// TIA Portal V21 export
FUNCTION "Motore_CentrifugaLavaggio" : Void   // FC135, LAD
{ S7_Optimized_Access := 'TRUE' }
// stored: SetENOAutomatically false
   VAR_TEMP
      AutoPos : Bool;
      AutoNeg : Bool;
   END_VAR
BEGIN

REGION Network 1: Comando positivo in automatico
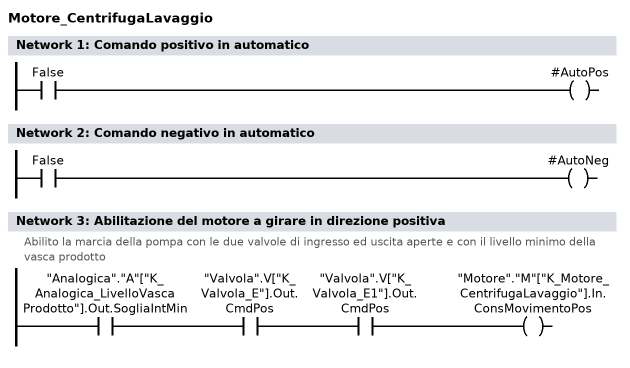
   RUNG wire#powerrail
      Contact( False )
      Coil( #AutoPos )
   END_RUNG
   // the same network as SCL:
   #AutoPos := False;
END_REGION

REGION Network 2: Comando negativo in automatico
   RUNG wire#powerrail
      Contact( False )
      Coil( #AutoNeg )
   END_RUNG
   // the same network as SCL:
   #AutoNeg := False;
END_REGION

REGION Network 3: Abilitazione del motore a girare in direzione positiva
   // Abilito la marcia della pompa con le due valvole di ingresso ed uscita aperte e con il livello minimo della vasca prodotto
   RUNG wire#powerrail
      Contact( "Analogica"."A"["K_Analogica_LivelloVascaProdotto"].Out.SogliaIntMin )
      Contact( "Valvola".V["K_Valvola_E"].Out.CmdPos )
      Contact( "Valvola".V["K_Valvola_E1"].Out.CmdPos )
      Coil( "Motore"."M"["K_Motore_CentrifugaLavaggio"].In.ConsMovimentoPos )
   END_RUNG
   // the same network as SCL:
   "Motore"."M"["K_Motore_CentrifugaLavaggio"].In.ConsMovimentoPos := "Analogica"."A"["K_Analogica_LivelloVascaProdotto"].Out.SogliaIntMin AND "Valvola".V["K_Valvola_E"].Out.CmdPos AND "Valvola".V["K_Valvola_E1"].Out.CmdPos;
END_REGION

REGION Network 4 (SCL)
   REGION CentrifugaLavaggio
       REGION Ingressi
           "Motore".M[K_Motore_CentrifugaLavaggio].In.FbDigitali.TermicoIntervenuto := NOT "CentrifugaLavaggio_TermicoOk";
           "Motore".M[K_Motore_CentrifugaLavaggio].In.FbDigitali.FeedbackMarcia := "CentrifugaLavaggio_Marcia";
           // "Motore".M["K_Motore_CentrifugaLavaggio"].In.CmdPosRich := #AutoPos;
           // "Motore".M["K_Motore_CentrifugaLavaggio"].In.CmdNegRich := #AutoNeg;
       END_REGION ;
       REGION Gestione
           "GestMotore"(K_Motore := "K_Motore_CentrifugaLavaggio",
                        K_TipoMotore := "K_TipoMotore_Teleruttore1Dir",
                        K_Zona := "K_Zona_Sterilizzatore");
       END_REGION ;
       REGION Uscite
           "CentrifugaLavaggio_ComandoMarcia" := "Motore".M[K_Motore_CentrifugaLavaggio].Out.CmdPosMotore;
       END_REGION ;
   END_REGION ;
END_REGION
END_FUNCTION
